(* Logix 5000 project; controller SpineControl2 vendor 1 type 14 code 155 rev 20.12; software revision 20.01 *)

TASK MainTask (continuous, watchdog 500 ms) : MainProgram

MODULES
   Local : vendor 1 type 14 code 155 (PointIO 0, rev 20.12)
      Motor_Driver : vendor 1 type 37 code 28 (Ethernet 192.168.1.5, rev 1.1, MotionDiagnostics RPI 1 ms, MotionSync RPI 1 ms)
      Discrete_IO : Embedded (PointIO 1, rev 20.11, Output RPI 20 ms)
END_MODULES

TYPE sock_structure :   // A user-defined structure that specifies the address for the socket.
STRUCT
   Family : INT;   // Specify the address family. Must be 2
   Port : INT;   // Specify the local port number on which an application is listening and receiving, or set to 0 if you want the EtherNet/IP module to choose the local port number: • For TCP client operations, specify 0 unless you want a specific local port number.For TCP server communication, specify the port number on which to accept incoming connection requests. • For UDP, specify a local port number to receive datagrams on a specific port.
   Addr : DINT;   // Specify an IP address. Typically, set to 0 (any address)
END_STRUCT
END_TYPE

TYPE sock_type_Accept_Response :
STRUCT
   Instance : INT;
   Addr : sock_structure;
END_STRUCT
END_TYPE

TYPE sock_type_Open :
STRUCT
   Timeout : DINT;   // Specify the timeout in milliseconds.
   DestAddr : STRING;   // Specify an array of characters (maximum of 64) to define the destination of the connection. Specify either of these: • Hostname?port=xxxzaz • IPAddr?port=xxx For example, to specify an IP address, enter 10.88.81.10?port=2813
END_STRUCT
END_TYPE

TYPE sock_type_Read_Params :
STRUCT
   Timeout : DINT;
   BufLen : DINT;
END_STRUCT
END_TYPE

TYPE sock_type_Read_Response :
STRUCT
   FromAddr : sock_structure;
   bufLen : DINT;
   Buf : SINT[200];   // contains the number of bytes of data received. Buf SINT array Contains the data. This number must be large enough to contain the maximum amount of data expected. For a standard connection, the maximum is SINT[484]; for a large connection the maximum is SINT [3984].
END_STRUCT
END_TYPE

TYPE sock_type_Socket_Create :   // Data Type for Socket Create Source Element
STRUCT
   Type : DINT;   // 1 for TCP, 2 for UDP
   Addr : sock_structure;   // specifies the address for the socket
END_STRUCT
END_TYPE

TYPE sock_type_Write_Pram :
STRUCT
   Timeout : DINT;   // milliseconds
   ToAddr : sock_structure;
   BufLen : DINT;
   Buf : SINT[480];   // Data to send
END_STRUCT
END_TYPE

VAR_GLOBAL   (* controller tags *)
   Delete_All_MSG : MESSAGE;
        MessageParameters(ServiceCode := 16#0051, ...)
   Delete_All_Request : BOOL;
   m_Accel_Jerk : DINT := 1;
   m_Accel_Rate : DINT := 2;
   m_Calc_Data : DINT;
   m_Decel_Jerk : DINT := 1;
   m_Decel_Rate : DINT := 2;
   m_Event_Dist : DINT;
   m_Lock_Position : DINT;
   m_MAH : MOTION_INSTRUCTION := (FLAGS := 33554432);
   m_MAM : MOTION_INSTRUCTION := (FLAGS := 33554432);
   m_MSF : MOTION_INSTRUCTION := (FLAGS := 33554432);
   m_MSO : MOTION_INSTRUCTION := (FLAGS := 33554432);
   m_Position : DINT := 50;
   m_Speed : DINT := 5;
   m_Type : DINT;
   motor1 : AXIS_CIP_DRIVE;
   motor_Enable : BOOL;
   Motor_Group : MOTION_GROUP;
   move2Home : BOOL;
   sock_Accept_Connection : MESSAGE;
        MessageParameters(ServiceCode := 16#0050, LocalElement := Sock_Accept_Connection_Param, DestinationTag := Sock_Accept_Connection_Responce, ...)
   Sock_Accept_Connection_Param : DINT := 5000;
   Sock_Accept_Connection_Responce : sock_type_Accept_Response;
   sock_Create : MESSAGE;
        MessageParameters(ServiceCode := 16#004b, LocalElement := Sock_Create_Param, DestinationTag := Sock_Create_Return, ...)
   Sock_Create_Param : sock_type_Socket_Create := (Type := 1, Addr.Family := 2, Addr.Port := 20);   // the input parameters to creating a socket
   Sock_Create_Return : DINT := 27010;   // The return value of the sockCreate message
   sock_Read : MESSAGE;
        MessageParameters(ServiceCode := 16#004d, LocalElement := Sock_Read_Param, DestinationTag := Sock_Read_Responce, ...)
   Sock_Read_Param : sock_type_Read_Params;
   Sock_Read_Responce : sock_type_Read_Response;
   sock_Write : MESSAGE;
        MessageParameters(ServiceCode := 16#004e, LocalElement := Sock_Write_Param, DestinationTag := Sock_Write_Response, ...)
   Sock_Write_Param : sock_type_Write_Pram;
   Sock_Write_Response : DINT;
   start_Motion : BOOL;
   start_Socket : BOOL;
   stop : BOOL;
   test_output : BOOL;
   test_output_stage_1 : BOOL;
   wait : BOOL;
END_VAR

PROGRAM MainProgram   (* main routine MainRoutine *)

ROUTINE MainRoutine   (* ladder *)
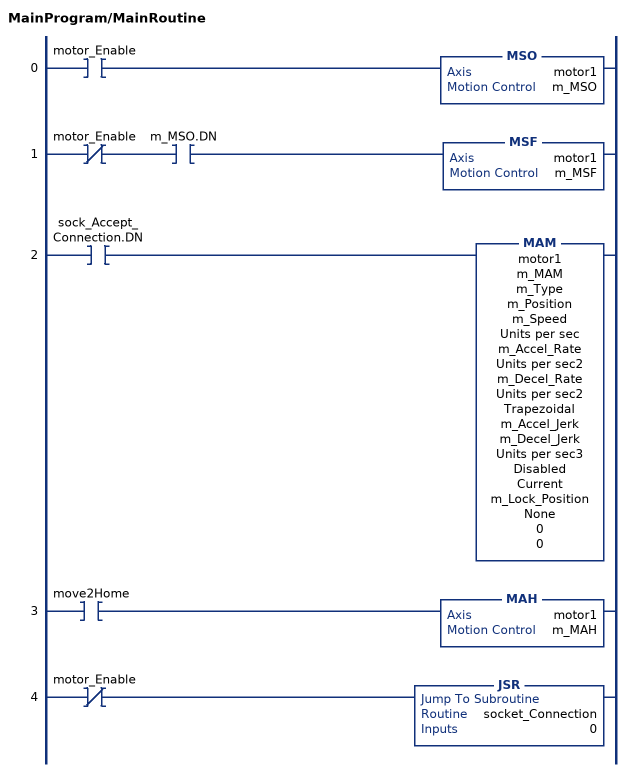
   0: XIC(motor_Enable)MSO(motor1,m_MSO);
   1: XIO(motor_Enable)XIC(m_MSO.DN)MSF(motor1,m_MSF);
   2: XIC(sock_Accept_Connection.DN)MAM(motor1,m_MAM,m_Type,m_Position,m_Speed,Units per sec,m_Accel_Rate,Units per sec2,m_Decel_Rate,Units per sec2,Trapezoidal,m_Accel_Jerk,m_Decel_Jerk,Units per sec3,Disabled,Current,m_Lock_Position,None,0,0);
   3: XIC(move2Home)MAH(motor1,m_MAH);
   4: XIO(motor_Enable)JSR(socket_Connection,0);
END_ROUTINE

ROUTINE socket_Connection   (* ladder *)
// TCP connection to c++ GUI
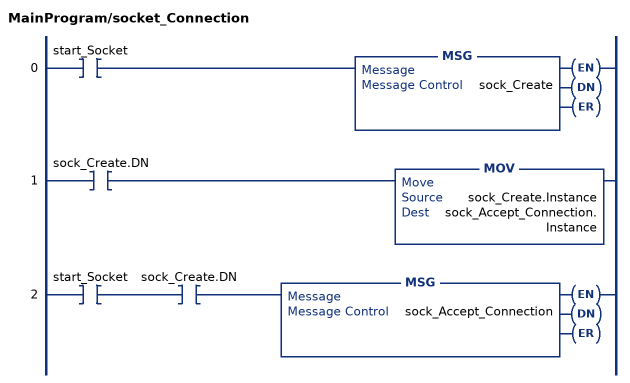
   0: XIC(start_Socket)MSG(sock_Create);
   1: XIC(sock_Create.DN)MOV(sock_Create.Instance,sock_Accept_Connection.Instance);
   2: XIC(start_Socket)XIC(sock_Create.DN)MSG(sock_Accept_Connection);
END_ROUTINE

ROUTINE socket_listener   (* ladder *)
// listen for incoming data
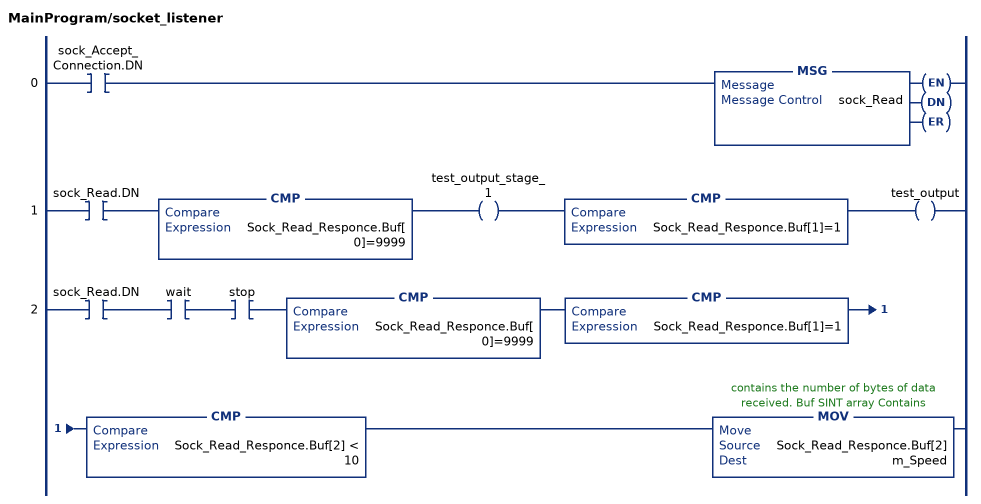
   0: XIC(sock_Accept_Connection.DN)MSG(sock_Read);
   1: XIC(sock_Read.DN)CMP(Sock_Read_Responce.Buf[0]=9999)OTE(test_output_stage_1)CMP(Sock_Read_Responce.Buf[1]=1)OTE(test_output);
   2: XIC(sock_Read.DN)XIC(wait)XIC(stop)CMP(Sock_Read_Responce.Buf[0]=9999)CMP(Sock_Read_Responce.Buf[1]=1)CMP(Sock_Read_Responce.Buf[2] < 10)MOV(Sock_Read_Responce.Buf[2],m_Speed);
END_ROUTINE
END_PROGRAM
